FUNCTION_BLOCK FB_Demarcate//CCD标定自动程序
VAR_INPUT
	AxisX1_NO : INT; //X1轴号
	AxisX2_NO : INT;//X2轴号
	AxisY_NO  : INT;//Y轴号	
END_VAR
VAR_OUTPUT
	
END_VAR
VAR
	
	i: INT;
	// 拍照延时复位
	TON1: TON;
	TON2: TON;
	// CCD标定上升沿
	rCCD_Demarcate: R_TRIG;
	singeMode: BOOL;
	singeStep0: BOOL;
	fCCD_Demarcate: F_TRIG;
	bTest1: BOOL;
	iTest: INT;
END_VAR

VAR_IN_OUT
	Step0: INT;//程序步
	DemarcateStart:BOOL;//CCD标定启动	
	CCDStart: BOOL;// CCD拍照启动
	CCDNo:INT;//ccd拍照次数记数
	DemarcateResult:INT;//标定结果
	DemarcateDone: BOOL;	// CCD标定完成
	Demarcateing: BOOL;	// CCD标定中
	// CCD标定NG报警
	Error: BOOL;
END_VAR

TON1(IN:= , PT:=T#2S , Q=> , ET=> );//拍照延时复位
TON2(IN:= , PT:=T#0.2S , Q=> , ET=> );//拍照延时
rCCD_Demarcate(CLK:=DemarcateStart , Q=> );//CCD标定启动上升沿
fCCD_Demarcate(CLK:=DemarcateStart , Q=> );//CCD标定启动上升沿
IF rCCD_Demarcate.Q THEN
	Error:=FALSE;//CCD标定NG报警
	TON1.IN:=FALSE;
	Step0:=0;
END_IF



CASE Step0 OF
		0://等待CCD标定启动信号
			IF fCCD_Demarcate.Q THEN
						i:=0;//标定点位记数
						TON1.IN:=FALSE;
						DemarcateStart:=FALSE;//复位标定启动
						DemarcateDone:=FALSE;//CCD标定完成
						Demarcateing:=TRUE;//CCD标定中
						IF singeMode THEN
							singeStep0:=TRUE;
						ELSE
							singeStep0:=FALSE;
						END_IF
						Step0:=10;
			END_IF
	10://X1、X2先回初始位
				IF  NOT singeStep0 THEN
							TON1.IN:=FALSE;
							IF arrAxisCtrl[AxisX1_NO].Status.Homed AND arrAxisCtrl[AxisX1_NO].Status.NoMoving THEN
										IF arrAxisCtrl[AxisX1_NO].Cmd.arrbRealPoint[1] THEN
											arrAxisCtrl[AxisX1_NO].Cmd.iGoSetPos:=0;
										ELSE
											arrAxisCtrl[AxisX1_NO].Cmd.iGoSetPos:=1;
										END_IF
							END_IF
							IF arrAxisCtrl[AxisX2_NO].Status.Homed AND arrAxisCtrl[AxisX2_NO].Status.NoMoving  THEN
										IF arrAxisCtrl[AxisX2_NO].Cmd.arrbRealPoint[1] THEN
											arrAxisCtrl[AxisX2_NO].Cmd.iGoSetPos:=0;
										ELSE
											arrAxisCtrl[AxisX2_NO].Cmd.iGoSetPos:=1;
										END_IF
							END_IF	
							IF  arrAxisCtrl[AxisX1_NO].Cmd.arrbRealPoint[1]  AND 	arrAxisCtrl[AxisX2_NO].Cmd.arrbRealPoint[1]THEN
								IF singeMode THEN
									singeStep0:=TRUE;
								ELSE
									singeStep0:=FALSE;
								END_IF
								Step0:=11;
							END_IF	
				END_IF		
	11://Y回初始位
				IF NOT singeStep0 THEN
									IF arrAxisCtrl[AxisY_NO].Status.Homed AND arrAxisCtrl[AxisY_NO].Status.NoMoving  THEN
											IF arrAxisCtrl[AxisY_NO].Cmd.arrbRealPoint[1] THEN
												arrAxisCtrl[AxisY_NO].Cmd.iGoSetPos:=0;
													IF singeMode THEN
														singeStep0:=TRUE;
													ELSE
														singeStep0:=FALSE;
													END_IF
													Step0:=12;									
											ELSE
												arrAxisCtrl[AxisY_NO].Cmd.iGoSetPos:=1;
											END_IF
								END_IF
				END_IF			
		12://判断CCD标定走到第几个点位
						IF NOT  singeStep0 THEN
											DemarcateResult:=0;
											IF  i=0    THEN//(-4,-4)
															arrAxisPar[AxisX1_NO].arrTargetPoint[3]:=arrAxisPar[AxisX1_NO].arrTargetPoint[1]-4;//+(103.94*COS(DEG_TO_RAD(CCD_W+225))-103.94*COS(DEG_TO_RAD(225))); 
															arrAxisPar[AxisX2_NO].arrTargetPoint[3]:=arrAxisPar[AxisX2_NO].arrTargetPoint[1]-4;//+(103.94*SIN(DEG_TO_RAD(CCD_W+315))-103.94*COS(DEG_TO_RAD(315)));
															arrAxisPar[AxisY_NO].arrTargetPoint[3]:=arrAxisPar[AxisY_NO].arrTargetPoint[1]-4;//+(103.94*COS(DEG_TO_RAD(CCD_W+135))-103.94*COS(DEG_TO_RAD(135)));	
															i:=i+1;
															IF singeMode THEN
																singeStep0:=TRUE;
															ELSE
																singeStep0:=FALSE;
															END_IF
															Step0:=20;
											ELSIF i=1 THEN//(0,-4)
															arrAxisPar[AxisX1_NO].arrTargetPoint[3]:=arrAxisPar[AxisX1_NO].arrTargetPoint[1];//+(103.94*COS(DEG_TO_RAD(CCD_W+225))-103.94*COS(DEG_TO_RAD(225))); 
															arrAxisPar[AxisX2_NO].arrTargetPoint[3]:=arrAxisPar[AxisX2_NO].arrTargetPoint[1];//+(103.94*SIN(DEG_TO_RAD(CCD_W+315))-103.94*COS(DEG_TO_RAD(315)));
															arrAxisPar[AxisY_NO].arrTargetPoint[3]:=arrAxisPar[AxisY_NO].arrTargetPoint[1]-4;//+(103.94*COS(DEG_TO_RAD(CCD_W+135))-103.94*COS(DEG_TO_RAD(135)));
															i:=i+1;
															IF singeMode THEN
																singeStep0:=TRUE;
															ELSE
																singeStep0:=FALSE;
															END_IF
															Step0:=20;
											ELSIF i=2 THEN//(4,-4)
															arrAxisPar[AxisX1_NO].arrTargetPoint[3]:=arrAxisPar[AxisX1_NO].arrTargetPoint[1]+4;//+(103.94*COS(DEG_TO_RAD(CCD_W+225))-103.94*COS(DEG_TO_RAD(225))); 
															arrAxisPar[AxisX2_NO].arrTargetPoint[3]:=arrAxisPar[AxisX2_NO].arrTargetPoint[1]+4;//+(103.94*SIN(DEG_TO_RAD(CCD_W+315))-103.94*COS(DEG_TO_RAD(315)));
															arrAxisPar[AxisY_NO].arrTargetPoint[3]:=arrAxisPar[AxisY_NO].arrTargetPoint[1]-4;//+(103.94*COS(DEG_TO_RAD(CCD_W+135))-103.94*COS(DEG_TO_RAD(135)));	
															i:=i+1;
															IF singeMode THEN
																singeStep0:=TRUE;
															ELSE
																singeStep0:=FALSE;
															END_IF
															Step0:=20;									
											ELSIF i=3 THEN//(4,0)
														arrAxisPar[AxisX1_NO].arrTargetPoint[3]:=arrAxisPar[AxisX1_NO].arrTargetPoint[1]+4;//+(103.94*COS(DEG_TO_RAD(CCD_W+225))-103.94*COS(DEG_TO_RAD(225))); 
														arrAxisPar[AxisX2_NO].arrTargetPoint[3]:=arrAxisPar[AxisX2_NO].arrTargetPoint[1]+4;//+(103.94*SIN(DEG_TO_RAD(CCD_W+315))-103.94*COS(DEG_TO_RAD(315)));
														arrAxisPar[AxisY_NO].arrTargetPoint[3]:=arrAxisPar[AxisY_NO].arrTargetPoint[1];//+(103.94*COS(DEG_TO_RAD(CCD_W+135))-103.94*COS(DEG_TO_RAD(135)));	
														i:=i+1;
														IF singeMode THEN
																singeStep0:=TRUE;
															ELSE
																singeStep0:=FALSE;
															END_IF
														Step0:=20;		
											ELSIF i=4 THEN//(0,0)
														arrAxisPar[AxisX1_NO].arrTargetPoint[3]:=arrAxisPar[AxisX1_NO].arrTargetPoint[1];//+(103.94*COS(DEG_TO_RAD(CCD_W+225))-103.94*COS(DEG_TO_RAD(225))); 
														arrAxisPar[AxisX2_NO].arrTargetPoint[3]:=arrAxisPar[AxisX2_NO].arrTargetPoint[1];//+(103.94*SIN(DEG_TO_RAD(CCD_W+315))-103.94*COS(DEG_TO_RAD(315)));
														arrAxisPar[AxisY_NO].arrTargetPoint[3]:=arrAxisPar[AxisY_NO].arrTargetPoint[1];//+(103.94*COS(DEG_TO_RAD(CCD_W+135))-103.94*COS(DEG_TO_RAD(135)));	
														i:=i+1;
														Step0:=20;		
											ELSIF i=5 THEN//(-4,0)
														arrAxisPar[AxisX1_NO].arrTargetPoint[3]:=arrAxisPar[AxisX1_NO].arrTargetPoint[1]-4;//+(103.94*COS(DEG_TO_RAD(CCD_W+225))-103.94*COS(DEG_TO_RAD(225))); 
														arrAxisPar[AxisX2_NO].arrTargetPoint[3]:=arrAxisPar[AxisX2_NO].arrTargetPoint[1]-4;//+(103.94*SIN(DEG_TO_RAD(CCD_W+315))-103.94*COS(DEG_TO_RAD(315)));
														arrAxisPar[AxisY_NO].arrTargetPoint[3]:=arrAxisPar[AxisY_NO].arrTargetPoint[1];//+(103.94*COS(DEG_TO_RAD(CCD_W+135))-103.94*COS(DEG_TO_RAD(135)));	
														i:=i+1;
														IF singeMode THEN
																singeStep0:=TRUE;
															ELSE
																singeStep0:=FALSE;
															END_IF
														Step0:=20;		
											ELSIF i=6 THEN//(-4,4)
															arrAxisPar[AxisX1_NO].arrTargetPoint[3]:=arrAxisPar[AxisX1_NO].arrTargetPoint[1]-4;//+(103.94*COS(DEG_TO_RAD(CCD_W+225))-103.94*COS(DEG_TO_RAD(225))); 
															arrAxisPar[AxisX2_NO].arrTargetPoint[3]:=arrAxisPar[AxisX2_NO].arrTargetPoint[1]-4;//+(103.94*SIN(DEG_TO_RAD(CCD_W+315))-103.94*COS(DEG_TO_RAD(315)));
															arrAxisPar[AxisY_NO].arrTargetPoint[3]:=arrAxisPar[AxisY_NO].arrTargetPoint[1]+4;//+(103.94*COS(DEG_TO_RAD(CCD_W+135))-103.94*COS(DEG_TO_RAD(135)));
															i:=i+1;
															IF singeMode THEN
																singeStep0:=TRUE;
															ELSE
																singeStep0:=FALSE;
															END_IF
															Step0:=20;		
											ELSIF i=7 THEN//(0,4)
															arrAxisPar[AxisX1_NO].arrTargetPoint[3]:=arrAxisPar[AxisX1_NO].arrTargetPoint[1];//+(103.94*COS(DEG_TO_RAD(CCD_W+225))-103.94*COS(DEG_TO_RAD(225))); 
															arrAxisPar[AxisX2_NO].arrTargetPoint[3]:=arrAxisPar[AxisX2_NO].arrTargetPoint[1];//+(103.94*SIN(DEG_TO_RAD(CCD_W+315))-103.94*COS(DEG_TO_RAD(315)));
															arrAxisPar[AxisY_NO].arrTargetPoint[3]:=arrAxisPar[AxisY_NO].arrTargetPoint[1]+4;//+(103.94*COS(DEG_TO_RAD(CCD_W+135))-103.94*COS(DEG_TO_RAD(135)));	
															i:=i+1;
															IF singeMode THEN
																singeStep0:=TRUE;
															ELSE
																singeStep0:=FALSE;
															END_IF
															Step0:=20;		
											ELSIF i=8 THEN//(4,4)
														arrAxisPar[AxisX1_NO].arrTargetPoint[3]:=arrAxisPar[AxisX1_NO].arrTargetPoint[1]+4;//+(103.94*COS(DEG_TO_RAD(CCD_W+225))-103.94*COS(DEG_TO_RAD(225))); 
														arrAxisPar[AxisX2_NO].arrTargetPoint[3]:=arrAxisPar[AxisX2_NO].arrTargetPoint[1]+4;//+(103.94*SIN(DEG_TO_RAD(CCD_W+315))-103.94*COS(DEG_TO_RAD(315)));
														arrAxisPar[AxisY_NO].arrTargetPoint[3]:=arrAxisPar[AxisY_NO].arrTargetPoint[1]+4;//+(103.94*COS(DEG_TO_RAD(CCD_W+135))-103.94*COS(DEG_TO_RAD(135)));	
														i:=i+1;
														IF singeMode THEN
																singeStep0:=TRUE;
															ELSE
																singeStep0:=FALSE;
															END_IF
														Step0:=20;		
											ELSIF i=9 THEN//(0,0,-2)
														arrAxisPar[AxisX1_NO].arrTargetPoint[3]:=arrAxisPar[AxisX1_NO].arrTargetPoint[1]+(103.94*COS(DEG_TO_RAD(-2+225))-103.94*COS(DEG_TO_RAD(225))); 
														arrAxisPar[AxisX2_NO].arrTargetPoint[3]:=arrAxisPar[AxisX2_NO].arrTargetPoint[1]+(103.94*COS(DEG_TO_RAD(-2+135))-103.94*COS(DEG_TO_RAD(135)));
														arrAxisPar[AxisY_NO].arrTargetPoint[3]:=arrAxisPar[AxisY_NO].arrTargetPoint[1]+(103.94*SIN(DEG_TO_RAD(-2+315))-103.94*SIN(DEG_TO_RAD(315)));	
														i:=i+1;
														IF singeMode THEN
																singeStep0:=TRUE;
															ELSE
																singeStep0:=FALSE;
															END_IF
														Step0:=20;		
											ELSIF i=10 THEN//(0,0)
														arrAxisPar[AxisX1_NO].arrTargetPoint[3]:=arrAxisPar[AxisX1_NO].arrTargetPoint[1];//+(103.94*COS(DEG_TO_RAD(2+225))-103.94*COS(DEG_TO_RAD(225))); 
														arrAxisPar[AxisX2_NO].arrTargetPoint[3]:=arrAxisPar[AxisX2_NO].arrTargetPoint[1];//+(103.94*SIN(DEG_TO_RAD(2+315))-103.94*COS(DEG_TO_RAD(315)));
														arrAxisPar[AxisY_NO].arrTargetPoint[3]:=arrAxisPar[AxisY_NO].arrTargetPoint[1];//+(103.94*COS(DEG_TO_RAD(2+135))-103.94*COS(DEG_TO_RAD(135)));	
														i:=i+1;
														IF singeMode THEN
																singeStep0:=TRUE;
															ELSE
																singeStep0:=FALSE;
															END_IF
														Step0:=20;		
											ELSIF i=11  THEN//(0,0,2)
															arrAxisPar[AxisX1_NO].arrTargetPoint[3]:=arrAxisPar[AxisX1_NO].arrTargetPoint[1]+(103.94*COS(DEG_TO_RAD(2+225))-103.94*COS(DEG_TO_RAD(225))); 
															arrAxisPar[AxisX2_NO].arrTargetPoint[3]:=arrAxisPar[AxisX2_NO].arrTargetPoint[1]+(103.94*COS(DEG_TO_RAD(2+135))-103.94*COS(DEG_TO_RAD(135)));
															arrAxisPar[AxisY_NO].arrTargetPoint[3]:=arrAxisPar[AxisY_NO].arrTargetPoint[1]+(103.94*SIN(DEG_TO_RAD(2+315))-103.94*SIN(DEG_TO_RAD(315)));
															i:=i+1;
															IF singeMode THEN
																singeStep0:=TRUE;
															ELSE
																singeStep0:=FALSE;
															END_IF
															Step0:=20;		
											ELSIF i=130 THEN
															arrAxisPar[AxisX1_NO].arrTargetPoint[3]:=arrAxisPar[AxisX1_NO].arrTargetPoint[1];//+(103.94*COS(DEG_TO_RAD(CCD_W+225))-103.94*COS(DEG_TO_RAD(225))); 
															arrAxisPar[AxisX2_NO].arrTargetPoint[3]:=arrAxisPar[AxisX2_NO].arrTargetPoint[1];//+(103.94*SIN(DEG_TO_RAD(CCD_W+315))-103.94*COS(DEG_TO_RAD(315)));
															arrAxisPar[AxisY_NO].arrTargetPoint[3]:=arrAxisPar[AxisY_NO].arrTargetPoint[1];//+(103.94*COS(DEG_TO_RAD(CCD_W+135))-103.94*COS(DEG_TO_RAD(135)));	
															i:=i+1;
															IF singeMode THEN
																singeStep0:=TRUE;
															ELSE
																singeStep0:=FALSE;
															END_IF
															Step0:=20;		
											ELSIF i=140 THEN
														arrAxisPar[AxisX1_NO].arrTargetPoint[3]:=arrAxisPar[AxisX1_NO].arrTargetPoint[1]+(103.94*COS(DEG_TO_RAD(-1+225))-103.94*COS(DEG_TO_RAD(225))); 
														arrAxisPar[AxisX2_NO].arrTargetPoint[3]:=arrAxisPar[AxisX2_NO].arrTargetPoint[1]+(103.94*SIN(DEG_TO_RAD(-1+315))-103.94*COS(DEG_TO_RAD(315)));
														arrAxisPar[AxisY_NO].arrTargetPoint[3]:=arrAxisPar[AxisY_NO].arrTargetPoint[1]+(103.94*COS(DEG_TO_RAD(-1+135))-103.94*COS(DEG_TO_RAD(135)));	
														i:=i+1;
														IF singeMode THEN
																singeStep0:=TRUE;
															ELSE
																singeStep0:=FALSE;
															END_IF
														Step0:=20;		
											ELSIF i=150 THEN
														arrAxisPar[AxisX1_NO].arrTargetPoint[3]:=arrAxisPar[AxisX1_NO].arrTargetPoint[1]+(103.94*COS(DEG_TO_RAD(-2+225))-103.94*COS(DEG_TO_RAD(225))); 
														arrAxisPar[AxisX2_NO].arrTargetPoint[3]:=arrAxisPar[AxisX2_NO].arrTargetPoint[1]+(103.94*SIN(DEG_TO_RAD(-2+315))-103.94*COS(DEG_TO_RAD(315)));
														arrAxisPar[AxisY_NO].arrTargetPoint[3]:=arrAxisPar[AxisY_NO].arrTargetPoint[1]+(103.94*COS(DEG_TO_RAD(-2+135))-103.94*COS(DEG_TO_RAD(135)));	
														i:=i+1;
														IF singeMode THEN
																singeStep0:=TRUE;
															ELSE
																singeStep0:=FALSE;
															END_IF
														Step0:=20;		
											ELSIF i=160 THEN
														arrAxisPar[AxisX1_NO].arrTargetPoint[3]:=arrAxisPar[AxisX1_NO].arrTargetPoint[1];//+(103.94*COS(DEG_TO_RAD(CCD_W+225))-103.94*COS(DEG_TO_RAD(225))); 
														arrAxisPar[AxisX2_NO].arrTargetPoint[3]:=arrAxisPar[AxisX2_NO].arrTargetPoint[1];//+(103.94*SIN(DEG_TO_RAD(CCD_W+315))-103.94*COS(DEG_TO_RAD(315)));
														arrAxisPar[AxisY_NO].arrTargetPoint[3]:=arrAxisPar[AxisY_NO].arrTargetPoint[1];//+(103.94*COS(DEG_TO_RAD(CCD_W+135))-103.94*COS(DEG_TO_RAD(135)));		
														i:=i+1;
														Step0:=20;													
											END_IF
						END_IF	
	20://先移动X1,X2
				IF  NOT singeStep0 THEN
					IF NOT TON1.Q THEN
										TON1.IN:=TRUE;
					ELSE
										IF arrAxisCtrl[AxisX1_NO].Status.Homed AND arrAxisCtrl[AxisX1_NO].Status.NoMoving THEN
													IF arrAxisCtrl[AxisX1_NO].Cmd.arrbRealPoint[3] THEN
														arrAxisCtrl[AxisX1_NO].Cmd.iGoSetPos:=0;
													ELSE
														arrAxisCtrl[AxisX1_NO].Cmd.iGoSetPos:=3;
													END_IF
										END_IF
										IF arrAxisCtrl[AxisX2_NO].Status.Homed AND arrAxisCtrl[AxisX2_NO].Status.NoMoving  THEN
													IF arrAxisCtrl[AxisX2_NO].Cmd.arrbRealPoint[3] THEN
														arrAxisCtrl[AxisX2_NO].Cmd.iGoSetPos:=0;
													ELSE
														arrAxisCtrl[AxisX2_NO].Cmd.iGoSetPos:=3;
													END_IF
										END_IF	
										IF  arrAxisCtrl[AxisX1_NO].Cmd.arrbRealPoint[3]  AND arrAxisCtrl[AxisX1_NO].Status.NoMoving AND 
							 				arrAxisCtrl[AxisX2_NO].Cmd.arrbRealPoint[3] AND arrAxisCtrl[AxisX2_NO].Status.NoMoving THEN
													IF singeMode THEN
														singeStep0:=TRUE;
													ELSE
														singeStep0:=FALSE;
													END_IF
													TON1.IN:=FALSE;
													Step0:=30;
										ELSIF arrAxisCtrl[AxisX1_NO].Status.Error OR arrAxisCtrl[AxisX2_NO].Status.Error THEN
													TON1.IN:=FALSE;
													Step0:=0;											
										END_IF	
						END_IF
				END_IF	
	30://再移动Y
				IF NOT singeStep0 THEN
							IF NOT TON1.Q THEN
										TON1.IN:=TRUE;
							ELSE
									IF arrAxisCtrl[AxisY_NO].Status.Homed AND arrAxisCtrl[AxisY_NO].Status.NoMoving  THEN
												IF arrAxisCtrl[AxisY_NO].Cmd.arrbRealPoint[3] THEN
													arrAxisCtrl[AxisY_NO].Cmd.iGoSetPos:=0;
														IF singeMode THEN
															singeStep0:=TRUE;
														ELSE
															singeStep0:=FALSE;
														END_IF
														TON1.IN:=FALSE;
														 TON2.IN:=FALSE;
														Step0:=31;									
												ELSE
													arrAxisCtrl[AxisY_NO].Cmd.iGoSetPos:=3;
												END_IF
								ELSIF   arrAxisCtrl[AxisY_NO].Status.Error THEN
														TON1.IN:=FALSE;
														Step0:=0;										
								END_IF
							END_IF
				END_IF
				
	31:
	    TON2.IN:=TRUE;
		IF TON2.Q THEN
				CCDNo:=i;
				CCDStart:=TRUE;
				DemarcateResult:=0;	
				Step0:=40;	
				 TON2.IN:=FALSE;
		END_IF		 
	40://启动拍照
			IF NOT TON1.Q THEN
				TON1.IN:=TRUE;
			ELSE
				TON1.IN:=FALSE;	
				CCDStart:=FALSE;
				Step0:=50;
			END_IF
	50://等待标定结果
			IF DemarcateResult=1 THEN
				DemarcateResult:=0; 
				 Step0:=60;
			ELSE
				Error:=TRUE;//CCD标定NG报警
				Step0:=9999;
			END_IF
	60://判断标定次数
			IF i>=12 THEN
				Step0:=0;
				Demarcateing:=FALSE;
			ELSE
				Step0:=10;
			END_IF				
END_CASE







IF bTest1 THEN
	
   CASE iTest OF
	 0://(-4,-4)
				arrAxisPar[AxisX1_NO].arrTargetPoint[3]:=arrAxisPar[AxisX1_NO].arrTargetPoint[1]-4;//+(103.94*COS(DEG_TO_RAD(CCD_W+225))-103.94*COS(DEG_TO_RAD(225))); 
				arrAxisPar[AxisX2_NO].arrTargetPoint[3]:=arrAxisPar[AxisX2_NO].arrTargetPoint[1]-4;//+(103.94*SIN(DEG_TO_RAD(CCD_W+315))-103.94*COS(DEG_TO_RAD(315)));
				arrAxisPar[AxisY_NO].arrTargetPoint[3]:=arrAxisPar[AxisY_NO].arrTargetPoint[1]-4;//+(103.94*COS(DEG_TO_RAD(CCD_W+135))-103.94*COS(DEG_TO_RAD(135)));	
				iTest:=50;
											
	 1://(0,-4)
			arrAxisPar[AxisX1_NO].arrTargetPoint[3]:=arrAxisPar[AxisX1_NO].arrTargetPoint[1];//+(103.94*COS(DEG_TO_RAD(CCD_W+225))-103.94*COS(DEG_TO_RAD(225))); 
		    arrAxisPar[AxisX2_NO].arrTargetPoint[3]:=arrAxisPar[AxisX2_NO].arrTargetPoint[1];//+(103.94*SIN(DEG_TO_RAD(CCD_W+315))-103.94*COS(DEG_TO_RAD(315)));
			arrAxisPar[AxisY_NO].arrTargetPoint[3]:=arrAxisPar[AxisY_NO].arrTargetPoint[1]-4;//+(103.94*COS(DEG_TO_RAD(CCD_W+135))-103.94*COS(DEG_TO_RAD(135)));
				iTest:=50;											
	2://(4,-4)
			arrAxisPar[AxisX1_NO].arrTargetPoint[3]:=arrAxisPar[AxisX1_NO].arrTargetPoint[1]+4;//+(103.94*COS(DEG_TO_RAD(CCD_W+225))-103.94*COS(DEG_TO_RAD(225))); 
			arrAxisPar[AxisX2_NO].arrTargetPoint[3]:=arrAxisPar[AxisX2_NO].arrTargetPoint[1]+4;//+(103.94*SIN(DEG_TO_RAD(CCD_W+315))-103.94*COS(DEG_TO_RAD(315)));
			arrAxisPar[AxisY_NO].arrTargetPoint[3]:=arrAxisPar[AxisY_NO].arrTargetPoint[1]-4;//+(103.94*COS(DEG_TO_RAD(CCD_W+135))-103.94*COS(DEG_TO_RAD(135)));	
				iTest:=50;															
	3://(4,0)
			arrAxisPar[AxisX1_NO].arrTargetPoint[3]:=arrAxisPar[AxisX1_NO].arrTargetPoint[1]+4;//+(103.94*COS(DEG_TO_RAD(CCD_W+225))-103.94*COS(DEG_TO_RAD(225))); 
			arrAxisPar[AxisX2_NO].arrTargetPoint[3]:=arrAxisPar[AxisX2_NO].arrTargetPoint[1]+4;//+(103.94*SIN(DEG_TO_RAD(CCD_W+315))-103.94*COS(DEG_TO_RAD(315)));
			arrAxisPar[AxisY_NO].arrTargetPoint[3]:=arrAxisPar[AxisY_NO].arrTargetPoint[1];//+(103.94*COS(DEG_TO_RAD(CCD_W+135))-103.94*COS(DEG_TO_RAD(135)));	
			iTest:=50;								
  4://(0,0)
		arrAxisPar[AxisX1_NO].arrTargetPoint[3]:=arrAxisPar[AxisX1_NO].arrTargetPoint[1];//+(103.94*COS(DEG_TO_RAD(CCD_W+225))-103.94*COS(DEG_TO_RAD(225))); 
		arrAxisPar[AxisX2_NO].arrTargetPoint[3]:=arrAxisPar[AxisX2_NO].arrTargetPoint[1];//+(103.94*SIN(DEG_TO_RAD(CCD_W+315))-103.94*COS(DEG_TO_RAD(315)));
			arrAxisPar[AxisY_NO].arrTargetPoint[3]:=arrAxisPar[AxisY_NO].arrTargetPoint[1];//+(103.94*COS(DEG_TO_RAD(CCD_W+135))-103.94*COS(DEG_TO_RAD(135)));	
			iTest:=50;
5://(-4,0)
			arrAxisPar[AxisX1_NO].arrTargetPoint[3]:=arrAxisPar[AxisX1_NO].arrTargetPoint[1]-4;//+(103.94*COS(DEG_TO_RAD(CCD_W+225))-103.94*COS(DEG_TO_RAD(225))); 
			arrAxisPar[AxisX2_NO].arrTargetPoint[3]:=arrAxisPar[AxisX2_NO].arrTargetPoint[1]-4;//+(103.94*SIN(DEG_TO_RAD(CCD_W+315))-103.94*COS(DEG_TO_RAD(315)));
		arrAxisPar[AxisY_NO].arrTargetPoint[3]:=arrAxisPar[AxisY_NO].arrTargetPoint[1];//+(103.94*COS(DEG_TO_RAD(CCD_W+135))-103.94*COS(DEG_TO_RAD(135)));	
		iTest:=50;
6://(-4,4)
			arrAxisPar[AxisX1_NO].arrTargetPoint[3]:=arrAxisPar[AxisX1_NO].arrTargetPoint[1]-4;//+(103.94*COS(DEG_TO_RAD(CCD_W+225))-103.94*COS(DEG_TO_RAD(225))); 
			arrAxisPar[AxisX2_NO].arrTargetPoint[3]:=arrAxisPar[AxisX2_NO].arrTargetPoint[1]-4;//+(103.94*SIN(DEG_TO_RAD(CCD_W+315))-103.94*COS(DEG_TO_RAD(315)));
			arrAxisPar[AxisY_NO].arrTargetPoint[3]:=arrAxisPar[AxisY_NO].arrTargetPoint[1]+4;//+(103.94*COS(DEG_TO_RAD(CCD_W+135))-103.94*COS(DEG_TO_RAD(135)));
			iTest:=50;										
7://(0,4)
		arrAxisPar[AxisX1_NO].arrTargetPoint[3]:=arrAxisPar[AxisX1_NO].arrTargetPoint[1];//+(103.94*COS(DEG_TO_RAD(CCD_W+225))-103.94*COS(DEG_TO_RAD(225))); 
		arrAxisPar[AxisX2_NO].arrTargetPoint[3]:=arrAxisPar[AxisX2_NO].arrTargetPoint[1];//+(103.94*SIN(DEG_TO_RAD(CCD_W+315))-103.94*COS(DEG_TO_RAD(315)));
		arrAxisPar[AxisY_NO].arrTargetPoint[3]:=arrAxisPar[AxisY_NO].arrTargetPoint[1]+4;//+(103.94*COS(DEG_TO_RAD(CCD_W+135))-103.94*COS(DEG_TO_RAD(135)));	
			iTest:=50;									
8://(4,4)
		arrAxisPar[AxisX1_NO].arrTargetPoint[3]:=arrAxisPar[AxisX1_NO].arrTargetPoint[1]+4;//+(103.94*COS(DEG_TO_RAD(CCD_W+225))-103.94*COS(DEG_TO_RAD(225))); 
			arrAxisPar[AxisX2_NO].arrTargetPoint[3]:=arrAxisPar[AxisX2_NO].arrTargetPoint[1]+4;//+(103.94*SIN(DEG_TO_RAD(CCD_W+315))-103.94*COS(DEG_TO_RAD(315)));
		arrAxisPar[AxisY_NO].arrTargetPoint[3]:=arrAxisPar[AxisY_NO].arrTargetPoint[1]+4;//+(103.94*COS(DEG_TO_RAD(CCD_W+135))-103.94*COS(DEG_TO_RAD(135)));	
		iTest:=50;
9://(0,0,-2)
			arrAxisPar[AxisX1_NO].arrTargetPoint[3]:=arrAxisPar[AxisX1_NO].arrTargetPoint[1]+(103.94*COS(DEG_TO_RAD(-2+225))-103.94*COS(DEG_TO_RAD(225))); 
				arrAxisPar[AxisX2_NO].arrTargetPoint[3]:=arrAxisPar[AxisX2_NO].arrTargetPoint[1]+(103.94*COS(DEG_TO_RAD(-2+135))-103.94*COS(DEG_TO_RAD(135)));
		arrAxisPar[AxisY_NO].arrTargetPoint[3]:=arrAxisPar[AxisY_NO].arrTargetPoint[1]+(103.94*SIN(DEG_TO_RAD(-2+315))-103.94*SIN(DEG_TO_RAD(315)));	
		iTest:=50;
11://(0,0,2)
				arrAxisPar[AxisX1_NO].arrTargetPoint[3]:=arrAxisPar[AxisX1_NO].arrTargetPoint[1]+(103.94*COS(DEG_TO_RAD(2+225))-103.94*COS(DEG_TO_RAD(225))); 
	arrAxisPar[AxisX2_NO].arrTargetPoint[3]:=arrAxisPar[AxisX2_NO].arrTargetPoint[1]+(103.94*COS(DEG_TO_RAD(2+135))-103.94*COS(DEG_TO_RAD(135)));
		arrAxisPar[AxisY_NO].arrTargetPoint[3]:=arrAxisPar[AxisY_NO].arrTargetPoint[1]+(103.94*SIN(DEG_TO_RAD(2+315))-103.94*SIN(DEG_TO_RAD(315)));
		iTest:=50;
12:
		arrAxisPar[AxisX1_NO].arrTargetPoint[3]:=arrAxisPar[AxisX1_NO].arrTargetPoint[1]+(103.94*COS(DEG_TO_RAD(-1+225))-103.94*COS(DEG_TO_RAD(225))); 
			arrAxisPar[AxisX2_NO].arrTargetPoint[3]:=arrAxisPar[AxisX2_NO].arrTargetPoint[1]+(103.94*SIN(DEG_TO_RAD(-1+315))-103.94*COS(DEG_TO_RAD(315)));
			arrAxisPar[AxisY_NO].arrTargetPoint[3]:=arrAxisPar[AxisY_NO].arrTargetPoint[1]+(103.94*COS(DEG_TO_RAD(-1+135))-103.94*COS(DEG_TO_RAD(135)));	
		iTest:=50;											
13:
		arrAxisPar[AxisX1_NO].arrTargetPoint[3]:=arrAxisPar[AxisX1_NO].arrTargetPoint[1]+(103.94*COS(DEG_TO_RAD(-2+225))-103.94*COS(DEG_TO_RAD(225))); 
			arrAxisPar[AxisX2_NO].arrTargetPoint[3]:=arrAxisPar[AxisX2_NO].arrTargetPoint[1]+(103.94*SIN(DEG_TO_RAD(-2+315))-103.94*COS(DEG_TO_RAD(315)));
			arrAxisPar[AxisY_NO].arrTargetPoint[3]:=arrAxisPar[AxisY_NO].arrTargetPoint[1]+(103.94*COS(DEG_TO_RAD(-2+135))-103.94*COS(DEG_TO_RAD(135)));	
		iTest:=50;							
14:
		arrAxisPar[AxisX1_NO].arrTargetPoint[3]:=arrAxisPar[AxisX1_NO].arrTargetPoint[1];//+(103.94*COS(DEG_TO_RAD(CCD_W+225))-103.94*COS(DEG_TO_RAD(225))); 
			arrAxisPar[AxisX2_NO].arrTargetPoint[3]:=arrAxisPar[AxisX2_NO].arrTargetPoint[1];//+(103.94*SIN(DEG_TO_RAD(CCD_W+315))-103.94*COS(DEG_TO_RAD(315)));
		arrAxisPar[AxisY_NO].arrTargetPoint[3]:=arrAxisPar[AxisY_NO].arrTargetPoint[1];//+(103.94*COS(DEG_TO_RAD(CCD_W+135))-103.94*COS(DEG_TO_RAD(135)));		
		iTest:=50;			
   
  50:  //先移动X1,X2
		
									  IF arrAxisCtrl[AxisX1_NO].Status.Homed AND arrAxisCtrl[AxisX1_NO].Status.NoMoving THEN
													IF arrAxisCtrl[AxisX1_NO].Cmd.arrbRealPoint[3] THEN
														arrAxisCtrl[AxisX1_NO].Cmd.iGoSetPos:=0;
													ELSE
														arrAxisCtrl[AxisX1_NO].Cmd.iGoSetPos:=3;
													END_IF
										END_IF
										IF arrAxisCtrl[AxisX2_NO].Status.Homed AND arrAxisCtrl[AxisX2_NO].Status.NoMoving  THEN
													IF arrAxisCtrl[AxisX2_NO].Cmd.arrbRealPoint[3] THEN
														arrAxisCtrl[AxisX2_NO].Cmd.iGoSetPos:=0;
													ELSE
														arrAxisCtrl[AxisX2_NO].Cmd.iGoSetPos:=3;
													END_IF
										END_IF	
										IF  arrAxisCtrl[AxisX1_NO].Cmd.arrbRealPoint[3]  AND arrAxisCtrl[AxisX1_NO].Status.NoMoving AND 
							 				arrAxisCtrl[AxisX2_NO].Cmd.arrbRealPoint[3] AND arrAxisCtrl[AxisX2_NO].Status.NoMoving THEN
											iTest:=60;		
										END_IF	
				
	60://再移动Y
		
									IF arrAxisCtrl[AxisY_NO].Status.Homed AND arrAxisCtrl[AxisY_NO].Status.NoMoving  THEN
												IF arrAxisCtrl[AxisY_NO].Cmd.arrbRealPoint[3] THEN
													arrAxisCtrl[AxisY_NO].Cmd.iGoSetPos:=0;
									                  bTest1:=FALSE;
														iTest:=66;									
												ELSE
													arrAxisCtrl[AxisY_NO].Cmd.iGoSetPos:=3;
												END_IF
									
								END_IF
	
		
END_CASE

END_IF

END_FUNCTION_BLOCK

(* stored: Version 1.1.0.1, ProductVersion 3.1.4024.12
   POU FB_Demarcate: Id {c551e839-9915-4045-a832-d8c254136c19}, SpecialFunc None *)
